(* IEC 61131-3 sources: standardizer-tutorial-lib/src/ControlModules, 9 files *)

(* ---- IFillingLevel.st ---- *)
NAMESPACE Simatic.Ax.Tutorial
    INTERFACE IFillingLevel
        METHOD GetFillingLevel : LREAL END_METHOD
    END_INTERFACE
END_NAMESPACE

(* ---- IHeater.st ---- *)
NAMESPACE Simatic.Ax.Tutorial
    INTERFACE IHeater EXTENDS ISetPoint

        METHOD GetTemperature : LREAL
        END_METHOD

        METHOD Enable
        END_METHOD

        METHOD IsEnabled : BOOL
        END_METHOD

        METHOD Disable
        END_METHOD

    END_INTERFACE

END_NAMESPACE

(* ---- ISetpoint.st ---- *)
NAMESPACE Simatic.Ax.Tutorial
    INTERFACE ISetPoint
        METHOD SetSetpoint
            VAR_INPUT
                setpoint : LREAL;
            END_VAR
        END_METHOD

        METHOD GetSetpoint : LREAL
        END_METHOD

    END_INTERFACE

END_NAMESPACE

(* ---- FillingLevelAnalogValue.st ---- *)
USING Simatic.Ax.IO.Input;
NAMESPACE Simatic.Ax.Tutorial
    CLASS FillingLevelAnalogValue IMPLEMENTS IFillingLevel
        VAR PUBLIC
            Level : LRealInput;
        END_VAR

        METHOD PUBLIC GetFillingLevel : LREAL
            GetFillingLevel := Level.Q();
        END_METHOD
    END_CLASS

END_NAMESPACE

(* ---- FillingLevelConstValue.st ---- *)
NAMESPACE Simatic.Ax.Tutorial
    CLASS FillingLevelConstant500Liter IMPLEMENTS IFillingLevel
        VAR PUBLIC
            Level : LREAL := 500.0;
        END_VAR
        VAR PROTECTED

        END_VAR

        METHOD PUBLIC GetFillingLevel : LREAL
            GetFillingLevel := Level;
        END_METHOD
    END_CLASS

END_NAMESPACE

(* ---- HeatBlock.st ---- *)
USING Simatic.Ax.IO.Input;

NAMESPACE Simatic.Ax.Tutorial
    CLASS HeatBlock IMPLEMENTS IHeater
        VAR PUBLIC
            ActTemperature : LRealInput;
            TemperatureSp : SetpointBase;
        END_VAR
        VAR PROTECTED
            _isEnabled : BOOL;

        END_VAR

        METHOD PUBLIC Enable
            _isEnabled := TRUE;
        END_METHOD

        METHOD PUBLIC IsEnabled : BOOL
            IsEnabled := _isEnabled;
        END_METHOD

        METHOD PUBLIC Disable
            _isEnabled := FALSE;
        END_METHOD

        METHOD PUBLIC GetTemperature : LREAL
            GetTemperature := ActTemperature.Q();
        END_METHOD

        METHOD PUBLIC SetSetpoint
            VAR_INPUT
                setpoint : LREAL;
            END_VAR
            TemperatureSp.SetSetpoint(setpoint);
            ;
        END_METHOD

        METHOD PUBLIC GetSetpoint : LREAL
            GetSetpoint := TemperatureSp.GetSetpoint();
        END_METHOD
END_CLASS
END_NAMESPACE

(* ---- Mixer.st ---- *)
USING Simatic.Ax.Axis;
USING Simatic.Ax.Axis;
NAMESPACE Simatic.Ax.Tutorial
    CLASS Mixer
        VAR PRIVATE
            _motor : ISpeedAxis;
            _setpointSpeed : LREAL := 950.0;
            _direction : Direction := Direction#FORWARD;
        END_VAR

        METHOD PUBLIC ConnectMotor
            VAR_INPUT
                MotorInstance : ISpeedAxis;
            END_VAR
            _motor := MotorInstance;
        END_METHOD

        METHOD PUBLIC Enable
            _motor.MoveVelocity(Speed := _setpointSpeed, Direction := _direction);
        END_METHOD

        METHOD PUBLIC Disable
            _motor.Halt();
        END_METHOD

    END_CLASS

END_NAMESPACE

(* ---- SetpointBase.st ---- *)
NAMESPACE Simatic.Ax.Tutorial
    CLASS SetpointBase IMPLEMENTS ISetpoint
        VAR PUBLIC
            Value : LREAL;
        END_VAR
        VAR PROTECTED

        END_VAR

        METHOD PUBLIC SetSetpoint
            VAR_INPUT
                setpoint : LREAL;
            END_VAR
            Value := setpoint;
            ;
        END_METHOD

        METHOD PUBLIC GetSetpoint : LREAL
            GetSetpoint := Value;
        END_METHOD
    END_CLASS
END_NAMESPACE

(* ---- Tank.st ---- *)
NAMESPACE Simatic.Ax.Tutorial
    CLASS Tank
        VAR PUBLIC
            FillingLevel : IFillingLevel;
            CapacityLiters : LREAL;
        END_VAR
        VAR PROTECTED

        END_VAR

        /// This method returns the capacity of the tank
        METHOD PUBLIC GetCapacity : LREAL
            GetCapacity := CapacityLiters;
        END_METHOD

        METHOD PUBLIC ConnectFillingLevel
            VAR_INPUT
                ifl : IFillingLevel;
            END_VAR
            FillingLevel := ifl;
        END_METHOD

        METHOD PUBLIC GetFillingLevel : LREAL
            IF (FillingLevel <> NULL) THEN
                GetFillingLevel := FillingLevel.GetFillingLevel();
            ELSE
                GetFillingLevel := 0.0;
            END_IF;
        END_METHOD
        METHOD PUBLIC IsFull : BOOL
            IsFull := FillingLevel.GetFillingLevel() >= CapacityLiters - 1.0;
        END_METHOD

        METHOD PUBLIC IsEmpty : BOOL
            IsEmpty := FillingLevel.GetFillingLevel() < 1.0;
        END_METHOD
    END_CLASS
END_NAMESPACE
